{attribute 'tc_no_symbol'}
FUNCTION_BLOCK FB_ClientDataExcha
VAR_INPUT
	hSocket				: T_HSOCKET;
	aToServer			: ARRAY[1..MAX_PLCPRJ_RXBUFFER_SIZE] OF BYTE;//发送数据缓存区
	udiSendNumber : UDINT;
	xEnable: BOOL;//使能失效标志位
	xResetRequest: BOOL;   
	dwTimeOut: DWORD;//[ms],0 => no executing time limit
	xNeedReceive : BOOL;//检测是否需要接收标志位
	xReceiveAlways : BOOL ;//检测是否需要一直进行读取
END_VAR
VAR_OUTPUT
	xRdyCmd : BOOL;(*是否满足接收指令*)
	xDone: BOOL;(*完成条件满足*)
	xBusy: BOOL;(*动作正在执行*)
	xError: BOOL;(*错误条件满足*)
	udiErrorID: UDINT;(*错误码*)
	sFromServer		: T_MaxString;//实际接收数据(字符串)
	rxBuffer				: ARRAY[1..MAX_PLCPRJ_RXBUFFER_SIZE] OF BYTE;//接收缓存区域(byte数组)
END_VAR
VAR
{attribute 'tc_no_symbol'}
	eState: STATE;//当前状态
{attribute 'tc_no_symbol'}
	eClientState : E_ClientSteps;
{attribute 'tc_no_symbol'}
	xFirstInvocation: BOOL := TRUE;
{attribute 'tc_no_symbol'}	 
	xTimeOut: BOOL;
{attribute 'tc_no_symbol'}
	tOperationTimer : TON;
{attribute 'tc_no_symbol'}	
	fbSocketSend		: FB_SocketSend := ( tTimeout := PLCPRJ_RECEIVE_TIMEOUT );
{attribute 'tc_no_symbol'}
	fbSocketReceive		: FB_SocketReceive := ( tTimeout := PLCPRJ_RECEIVE_TIMEOUT );
{attribute 'tc_no_symbol'}
	fbReceiveTON		: TON;
{attribute 'tc_no_symbol'}	
	fbDisconnectTON		: TON;
{attribute 'tc_no_symbol'}
	RisingEdge			: R_TRIG;
{attribute 'tc_no_symbol'}	
	eDataExchaStep	: E_DataExchaSteps;
{attribute 'tc_no_symbol'}	
	cbReceived , idx	: UDINT;	
{attribute 'tc_no_symbol'}	
	_rxBufferTemp				: ARRAY[1..MAX_PLCPRJ_RXBUFFER_SIZE] OF BYTE;//接收缓存区域
{attribute 'tc_no_symbol'}	
_ton : TON;
END_VAR
VAR_TEMP
{attribute 'tc_no_symbol'}
	xAgain: BOOL;
END_VAR

xAgain:=0;

REPEAT
	CASE eState OF
		STATE.DORMANT:
				HandleDormantState(xAgain=> xAgain);
		STATE.EXECUTING:
				HandleExecutingState(xAgain=> xAgain);
		STATE.DONE:
				HandleDoneState(xAgain=> xAgain);
		STATE.INERROR:
				HandleErrorState(xAgain=> xAgain);
		STATE.ABORTING:
				HandleAbortingState(xAgain=> xAgain);
		STATE.RESETING:
				HandleResettingState(xAgain=> xAgain);
    END_CASE
UNTIL (xAgain=0)
END_REPEAT

xRdyCmd := 	eState = STATE.DORMANT;//输出是否已经准备好响应指令

{attribute 'tc_no_symbol'}
METHOD PROTECTED AbortAction
VAR_INPUT
END_VAR
VAR_OUTPUT
	xComplete: BOOL;
  udiErrorID: UDINT;
END_VAR
(*
* Cleaning
* => abort all running operation
* => if an UDINT codition is reached, set udiErrorID to a Value rather then 0 
*)
xComplete:=1;
udiErrorID:=0;
END_METHOD

{attribute 'tc_no_symbol'} 
METHOD PROTECTED CyclicAction
VAR_INPUT
END_VAR
VAR_OUTPUT
	xComplete: BOOL;
	udiErrorID: UDINT;
END_VAR
VAR	
END_VAR
{attribute 'tc_no_symbol'}
IF xFirstInvocation THEN
(*
* Staring
* for then first (!) invocaion,
* sample then input variables
*)		
	eDataExchaStep := DATAEXCHA_STATE_IDLE;
	xFirstInvocation:=0;			
END_IF    
REPEAT 	 
	CASE eDataExchaStep OF		
		DATAEXCHA_STATE_IDLE:						
			cbReceived := 0; // TODO. Leslie
			fbReceiveTON( IN := FALSE, PT := T#0s ); (* don't wait, read the first answer data immediately *)
			fbDisconnectTON( IN := FALSE, PT := T#0s );(* disable timeout check first *)
			eDataExchaStep := DATAEXCHA_STATE_SEND_START;
	   
		DATAEXCHA_STATE_SEND_START:
			fbSocketSend( bExecute := FALSE );
			fbSocketSend( 	hSocket	:= hSocket,
						cbLen	:= udiSendNumber,(* string length inclusive zero delimiter *)				
						pSrc	:= ADR( aToServer ),
						bExecute:= TRUE );//启动发送			
			eDataExchaStep := DATAEXCHA_STATE_SEND_WAIT;
	
		DATAEXCHA_STATE_SEND_WAIT:
			fbSocketSend( bExecute := FALSE );
			IF NOT fbSocketSend.bBusy THEN//检测发送是否完成
				IF NOT fbSocketSend.bError THEN	
					IF xNeedReceive
					THEN
						fbDisconnectTON(IN := FALSE);
						eDataExchaStep := DATAEXCHA_STATE_RECEIVE_START;							
					ELSE
						SysMemSet( ADR(sFromServer), 0, SIZEOF(sFromServer));		
						eDataExchaStep := DATAEXCHA_STATE_IDLE;		
						xComplete := 1;	
					END_IF	
				ELSE		
					udiErrorID := fbSocketSend.nErrId;								
				END_IF						
			END_IF		
	
		DATAEXCHA_STATE_RECEIVE_START:
			fbDisconnectTON(IN := TRUE,PT:=T#10MS);
			fbSocketReceive(bExecute := FALSE);		
			 
			fbSocketReceive(  hSocket:= hSocket,
											cbLen:= SIZEOF( _rxBufferTemp ),
											pDest:= ADR( _rxBufferTemp),
											bExecute:= TRUE ,
											nRecBytes=>cbReceived); 
      IF fbDisconnectTON.Q
			THEN
				eDataExchaStep := DATAEXCHA_STATE_RECEIVE_WAIT;
				fbDisconnectTON(IN:=FALSE);       
			END_IF
		DATAEXCHA_STATE_RECEIVE_WAIT:	
			_ton(IN:= NOT _ton.Q, PT:= T#20MS, Q=> , ET=> );
			fbSocketReceive(bExecute := _ton.Q,
                      nRecBytes=>cbReceived);	
      fbSocketReceive(bExecute := FALSE);				
			IF NOT fbSocketReceive.bBusy THEN
				IF NOT fbSocketReceive.bError THEN 						
					IF cbReceived < 255 AND cbReceived > 0 THEN(* no overflow *)
						fbReceiveTON( PT := T#0s ); (* bytes received => increase the read (polling) speed *)
						fbDisconnectTON( IN := FALSE );(* bytes received => disable timeout check *)		
						SysMemSet( ADR(sFromServer), 0, SIZEOF(sFromServer));		
						SysMemSet( ADR(rxBuffer), 0, SIZEOF(rxBuffer));	
						SysMemCpy( ADR( rxBuffer ), ADR( _rxBufferTemp ), cbReceived );//进行数据迁移
						SysMemCpy( ADR( sFromServer ), ADR( _rxBufferTemp ), cbReceived );(* copy the received string to the output variable (inclusive the end delimiter) *)								
						eDataExchaStep := DATAEXCHA_STATE_IDLE;		
						xComplete := 1;
					END_IF
					IF cbReceived >= 255(* there is no more free read buffer space => the answer string should be terminated *)	
          THEN
						udiErrorID :=100;(* buffer overflow !*)				
					END_IF			
				ELSE(* receive UDINT *)
					udiErrorID := fbSocketReceive.nErrId;	
				END_IF
			END_IF
			fbDisconnectTON( IN := TRUE, PT := PLCPRJ_RECEIVE_TIMEOUT );(* no bytes received => enable timeout check*)
			IF fbDisconnectTON.Q THEN (* timeout UDINT*)
				fbDisconnectTON( IN := FALSE );
				udiErrorID := 101;//接收超时报错			
			END_IF
		ELSE
			;
	END_CASE	       
UNTIL (TRUE)//让程序一直处于刷新状态
END_REPEAT

IF NOT xEnable OR xComplete OR udiErrorID<>0 THEN    
    (*
    * Cleaning
    * => free as much allocated resources as possible
    *)    
    tOperationTimer(IN:=0);
END_IF
END_METHOD

{attribute 'tc_no_symbol'}
METHOD PRIVATE FINAL HandleAbortingState
VAR_INPUT
END_VAR
VAR_OUTPUT
	xAgain: BOOL;
END_VAR
VAR
{attribute 'tc_no_symbol'}	
	xComplete: BOOL;
END_VAR
AbortAction(xComplete=> xComplete, udiErrorID=> udiErrorID);

IF udiErrorID<>0 THEN
    eState:=STATE.INERROR;
    xAgain:=1;
ELSIF xComplete THEN
    eState:=STATE.INERROR;
    xAgain:=1;
END_IF
END_METHOD

{attribute 'tc_no_symbol'}
METHOD PRIVATE FINAL HandleDoneState
VAR_INPUT
END_VAR
VAR_OUTPUT
	xAgain: BOOL;
END_VAR
IF xDone AND (xEnable=0) THEN
	eState:=STATE.RESETING;
	xAgain:=1;
ELSE
	xBusy:=0;
	xDone:=1;
	//xResetRequest:=(xExecute=0);
	xAgain:=0;(* !!! *)
END_IF
END_METHOD

{attribute 'tc_no_symbol'}
METHOD PRIVATE FINAL HandleDormantState
VAR_INPUT
END_VAR
VAR_OUTPUT
	xAgain: BOOL;
END_VAR
IF xEnable THEN
    xBusy:=1;
    eState:=STATE.EXECUTING;
    xAgain:=1;
END_IF
END_METHOD

{attribute 'tc_no_symbol'}
METHOD PRIVATE FINAL  HandleErrorState
VAR_INPUT
END_VAR
VAR_OUTPUT
	xAgain: BOOL;
END_VAR
IF xError AND (xResetRequest OR NOT xEnable ) THEN
    eState:=STATE.RESETING;
    xAgain:=1;
ELSE
    xBusy:=0;
    xError:=1;    
    xAgain:=0;(* !!! *)
END_IF
END_METHOD

{attribute 'tc_no_symbol'}
METHOD PRIVATE FINAL HandleExecutingState
VAR_INPUT
END_VAR
VAR_OUTPUT
	xAgain: BOOL;
END_VAR
VAR
{attribute 'tc_no_symbol'}	
	xComplete: BOOL;
END_VAR
 
CyclicAction(xComplete=> xComplete, udiErrorID=> udiErrorID);


IF udiErrorID<>0 THEN//检测是否有错误发生
    eState:=STATE.INERROR;
    xAgain:=1;
ELSIF NOT xEnable THEN//检测使能条件
    eState:=STATE.ABORTING;
    xAgain:=1;
ELSIF xComplete THEN//检测是否正常处理完成
    eState:=STATE.DONE;
    xAgain:=1;
END_IF
END_METHOD

{attribute 'tc_no_symbol'}
METHOD PRIVATE FINAL HandleResettingState
VAR_INPUT
END_VAR
VAR_OUTPUT
	xAgain: BOOL;
END_VAR
VAR
{attribute 'tc_no_symbol'}
	xComplete: BOOL;
END_VAR
ResetAction(xComplete=> xComplete);

IF xComplete THEN
		xEnable:=0;//清除输入指令 
    xBusy:=0;
    xDone:=0;
    xError:=0;

    udiErrorID:=0;
    eState:=STATE.DORMANT;
    xFirstInvocation:=1;
    xAgain:=0;(* !!! *)
END_IF
END_METHOD

{attribute 'tc_no_symbol'}
METHOD PROTECTED ResetAction
VAR_INPUT
END_VAR
VAR_OUTPUT
	xComplete: BOOL;
END_VAR
(*
* Cleaning
* => free all allocated resources
* => reinitialize instance variables
*)
tOperationTimer(IN:=0);

fbSocketSend( bExecute := FALSE );
fbSocketReceive(bExecute := FALSE);		

eDataExchaStep := DATAEXCHA_STATE_IDLE;		

xComplete := 1;
END_METHOD

END_FUNCTION_BLOCK

(* stored: Version 1.1.0.1, ProductVersion 3.1.4024.9
   POU FB_ClientDataExcha: Id {0e2a7d35-2b8a-47f0-8bf3-3aeafb69127f}, SpecialFunc None
   Method AbortAction: Id {16d50905-e8e6-4033-82bd-2d43d0f885af}
   Method CyclicAction: Id {fc8f39d9-2081-4e25-b3ae-b7fda8c58ea0}
   Method HandleAbortingState: Id {47b554fe-a5f2-448a-94d5-7d76d92ac5e7}
   Method HandleDoneState: Id {d72cccda-2d23-42ca-8362-5b60ad8fa845}
   Method HandleDormantState: Id {5128ac62-123d-4a36-bcd3-1f1e494b7c86}
   Method HandleErrorState: Id {12f672bd-2ef8-418b-9c73-7a7685022dfe}
   Method HandleExecutingState: Id {227577b8-e051-4fa2-9619-44166c8f0a11}
   Method HandleResettingState: Id {42ac0aa6-2380-423d-b54f-b9e577c1c3d2}
   Method ResetAction: Id {2eaba959-7737-4f6f-a06e-db29edecb0c1} *)
